// TwinCAT 3 PLC project LCLSGeneral
// Title: LCLS General
// Company: SLAC
// Author: Alex Wallace
// ProjectVersion: 0.0.0
// Description: Generally useful POUs: - Logger - FB diagnostics - EtherCAT diagnostic
// ProgramVersion: 3.1.4020.2
// libraries:
//   Tc2_EtherCAT, * (Beckhoff Automation GmbH)
//   Tc2_IoFunctions, * (Beckhoff Automation GmbH)
//   Tc2_ModbusSrv, * (Beckhoff Automation GmbH)
//   Tc2_SerialCom, * (Beckhoff Automation GmbH)
//   Tc2_Standard, * (Beckhoff Automation GmbH)
//   Tc2_System, * (Beckhoff Automation GmbH)
//   Tc2_TcpIp, * (Beckhoff Automation GmbH)
//   Tc2_Utilities, * (Beckhoff Automation GmbH)
//   Tc3_EventLogger, * (Beckhoff Automation GmbH)
//   Tc3_JsonXml, * (Beckhoff Automation GmbH)
//   Tc3_Module, * (Beckhoff Automation GmbH)
// project tree:
//   Data types/Misc/ ST_System.TcDUT (not stored)
//   GVLs/ DefaultGlobals.TcGVL (not stored), Global_Variables_EtherCAT.TcGVL (not stored)
//   Interfaces/ I_Interface.TcIO, I_Base.TcIO
//   POUs/Logger/ FB_LogHandler.TcPOU
//   / Task_3.TcTTO (not stored)

// ---- Interfaces/I_Interface.TcIO
INTERFACE I_Interface EXTENDS I_Base

VAR
	iVar1 : INT;
END_VAR
VAR_INPUT
	iInputVar1 : INT;
END_VAR
VAR_OUTPUT
	iOutputVar1 : INT;
END_VAR
VAR_EXTERNAL
	iExternVar1 : INT;
END_VAR

METHOD Method1 : BOOL
VAR_INPUT
END_VAR
END_METHOD

PROPERTY Property1 : INT
GET
END_GET
SET
END_SET
END_PROPERTY

END_INTERFACE

// ---- Interfaces/I_Base.TcIO
INTERFACE I_Base

VAR
	iTestBase : INT;
END_VAR

METHOD BaseMethod : BOOL
VAR_INPUT
END_VAR
END_METHOD

PROPERTY BaseProperty : INT
GET
END_GET
SET
END_SET
END_PROPERTY

END_INTERFACE

// ---- POUs/Logger/FB_LogHandler.TcPOU
FUNCTION_BLOCK FB_LogHandler
VAR_INPUT

	bLogHandlerInput : BOOL;

END_VAR

VAR CONSTANT
    nNumListeners		:	UINT	:= 6;
    DisarmCountDefault : UINT :=5; // # number of cycles to permit below threshold condition
END_VAR

ACTION CircuitBreaker:
// Global log circuit breaker
(*
Logic explanation
We want to trip if there is a constant stream of messages being emitted by this PLC. We also
only want the noisy offenders to trip. To target them we set a global trickle tripped flag
using this logic here. Then each individual FB_LogMessage evaluates itself to see if it's
sending a message too frequently (ie. it's being called to often).

This logic is attempting to implement the following:
1. Trip if the total events exceeds the nTrickleThreshold for >10s
2. Sustain the timer if the event count drops for a handful of cycles since usually a cycle amounts to 10ms, losing a few
should not stop the trickle timer.
*)
bTripCon := GVL_Logger.nGlobAccEvents >0;

tofTrickleBreakerPre(IN:=bTripCon);
tonTrickleBreaker(IN:=tofTrickleBreakerPre.Q);

GVL_Logger.bTrickleTripped S= tonTrickleBreaker.Q AND bTripCon;

GVL_Logger.nGlobAccEvents := 0; // reset the count for the next cycle
END_ACTION

END_FUNCTION_BLOCK
